(* IEC 61131-3 sources: go-native-ads/examples/rpc/plc/references, 3 files *)

(* ---- FillBuffer.st ---- *)
{attribute 'TcRpcEnable'}
METHOD PUBLIC FillBuffer
VAR_INPUT
    count : UINT;
END_VAR
VAR_OUTPUT
    {attribute 'TcRpcLengthIs' := 'count'}
    values : POINTER TO INT;
END_VAR
VAR
    i : UINT;
END_VAR

IF count > 0 AND values <> 0 THEN
    FOR i := 0 TO count - 1 DO
        values[i] := UINT_TO_INT(i * 2);
    END_FOR
END_IF

(* ---- Increment.st ---- *)
{attribute 'TcRpcEnable'}
METHOD PUBLIC Increment
VAR_IN_OUT
    value : DINT;
END_VAR

value := value + 1;

(* ---- SumBuffer.st ---- *)
{attribute 'TcRpcEnable'}
METHOD PUBLIC SumBuffer : DINT
VAR_INPUT
    count : UINT;
    {attribute 'TcRpcLengthIs' := 'count'}
    values : POINTER TO INT;
END_VAR
VAR
    i : UINT;
END_VAR

SumBuffer := 0;
IF count > 0 AND values <> 0 THEN
    FOR i := 0 TO count - 1 DO
        SumBuffer := SumBuffer + values[i];
    END_FOR
END_IF
